PROGRAM resetVars
VAR
END_VAR

//inputs
			GVL.filterPlaatsen := FALSE;
			GVL.waterreservoirVullen := FALSE;
			GVL.scoopieDrBij := FALSE;
			GVL.apparaatAanzetten := FALSE;
			GVL.ikBenMoe := FALSE;
			GVL.allesLegen := FALSE;
				
			//outputs
			GVL.apparaatAan := FALSE;
			GVL.filterGeplaatst := FALSE;
			GVL.aantalSchepjes := 0;
			GVL.reservoirLevel := 0;
			GVL.koffieKlaar := FALSE;
			GVL.apparaatLeeg := TRUE;
			GVL.koffieError := FALSE;
			GVL.waterigeKoffie := FALSE;
			GVL.sterkeKoffie := FALSE;
			GVL.lekkereKoffie := FALSE;

END_PROGRAM

(* stored: Version 1.1.0.1, ProductVersion 3.1.4024.12
   POU resetVars: Id {52921f20-f083-425f-80d1-3b4a69301866}, SpecialFunc None *)
